PROGRAM MAIN
VAR
	fbListenerTest : FB_ListenerTest;
END_VAR

fbListenerTest();

END_PROGRAM

(* stored: Version 1.1.0.1, ProductVersion 3.1.4022.10
   POU MAIN: Id {e5156229-dc7e-47cb-bfdc-7d4aa00249b1}, SpecialFunc None *)
